// TIA Portal V16 export
// export: Created 2021-11-12T13:32:17.1363904Z, ExportSetting WithDefaults, DisplayName Totally Integrated Automation Portal, DisplayVersion V16 Update 3, DisplayName TIA Portal Version Control Interface, DisplayVersion V16 Update 2, DisplayName TIA Portal Openness, DisplayVersion V16 Update 3, DisplayName SINAMICS Startdrive Advanced, DisplayVersion V16 Update 5, DisplayName SINAMICS Startdrive G130, G150, S120, S150, SINAMICS MV, S210, DisplayVersion V16 Update 5, DisplayName SINAMICS Startdrive G110M, G120, G120C, G120D, G120P, G115D, DisplayVersion V16 Update 5, DisplayName STEP 7 Professional, DisplayVersion V16 Update 3, DisplayName STEP 7 Safety, DisplayVersion V16, DisplayName WinCC UA Professional, DisplayVersion V16 Update 3
DATA_BLOCK "HMI_CMD_BSN2"   // DB34
{ S7_Optimized_Access := 'TRUE' }
VERSION : 0.1
// stored: AutoNumber true, DBAccessibleFromOPCUA true, IsOnlyStoredInLoadMemory false, IsRetainMemResEnabled false, IsWriteProtectedInAS false, MemoryReserve 100
   VAR
      Commands : "UDT_BSN_Command";   // Material flow commands
      xxxxx___Alarms___xxxxx : Byte;
      Furnace : "UDT_DI_Mon_Command";   // alarm from furnace
      LiveBit : "UDT_DI_Mon_Command";   // communication error
      DataTracking : "UDT_DI_Mon_Command";   // part on senzor is not in map
      Senzor : "UDT_DI_Mon_Command";   // part in map is not on senzor
      ProdParam : "UDT_DI_Mon_Command";   // production parameters have not changed
      "Step" : "UDT_DI_Mon_Command";   // long time without step
      Alarm_7 : "UDT_DI_Mon_Command";
   END_VAR
BEGIN
END_DATA_BLOCK
